FUNCTION_BLOCK SuccessTestRpcHandler IMPLEMENTS I_RpcHandler
VAR
END_VAR

METHOD Handle
VAR_INPUT
	Parameters : I_RpcParameters;
	Response : I_RpcResponse;
END_VAR
VAR
	fooParam : T_MAXSTRING;
	helloParam : T_MAXSTRING;
	result : T_MAXSTRING;
END_VAR
IF NOT Parameters.TryGetParameter('foo',fooParam) THEN
	Response.Reject('Missing foo parameter');
	RETURN;
END_IF

Parameters.TryGetParameter('hello',helloParam);

result := SuccessTestFunction(foo:=fooParam, hello:=helloParam);

Response.Build().StartObject().AddKeyString('test',result).EndObject().Finalize();

//Response.Reject('');
//Response.MakeAsync(myAsyncResponse);
END_METHOD

END_FUNCTION_BLOCK

(* stored: Version 1.1.0.1, ProductVersion 3.1.4024.12
   POU SuccessTestRpcHandler: Id {3308dee3-7162-4e6b-ab6c-6da43be8ef3f}, SpecialFunc None
   Method Handle: Id {b973a79f-d251-4a0d-baf6-50941936d5fe} *)
